FUNCTION_BLOCK EP7402_0xxx_Channel
VAR_INPUT
END_VAR
VAR_OUTPUT
END_VAR
VAR
	DI_Inputs AT%I* : DInputs;
	DO_Outputs AT%Q* : DOutputs;
	STM_Control AT%Q* : STMControl;
	STM_Info_data AT%I* : STMInfoData;
	STM_Input_Device AT%I* : STMInputDevice;
	STM_Status AT%I* : STMStatus;
	STM_Target_Velocity AT%Q* : STMTargetVelocity;
	
	_acceleration : UINT := 100;
	_deceleration : UINT := 100;
	
	State :(
		_00_mWait,
        _01_mReset,
        _02_mEnable,
		_03_mStop,
		_04_RunAtVelo,
		_05_mDisable);
		
	tonHoldHigh	: ton;
		
END_VAR

CASE State OF
        _00_mWait : 
			;
        _01_mReset : 
			STM_Control.reset := TRUE;
			tonHoldHigh(in := TRUE, pt := T#500MS);
			IF tonHoldHigh.Q THEN
				STM_Control.reset := FALSE;
				IF STM_Status.error = FALSE AND
					STM_Status.warning = FALSE AND
					STM_Status.ready = TRUE
				THEN
					State := _00_mWait;
					tonHoldHigh(in := FALSE);
				END_IF
			END_IF
			
        _02_mEnable : 
			IF STM_Status.error THEN				
				State := _01_mReset;
			ELSE
				STM_Control.enable := TRUE;			
			END_IF

			
		_04_RunAtVelo :
			;
			
		_03_mStop : 
			STM_Target_Velocity.velocity := 0;
			IF STM_Status.ready THEN	
				State := _02_mEnable;
			END_IF
			
		_05_mDisable:
			STM_Control.enable := FALSE;
			State := _00_mWait;
		
			
END_CASE

PROPERTY PUBLIC Acceleration : uint
GET
Acceleration := _acceleration;
END_GET
SET
_acceleration := Acceleration;
END_SET
END_PROPERTY

PROPERTY PUBLIC Deceleration : uint
GET
Deceleration := _deceleration;
END_GET
SET
_deceleration := Deceleration;
END_SET
END_PROPERTY

METHOD Disable : BOOL
VAR_INPUT
END_VAR
IF STM_Status.ready THEN
	State := _05_mDisable;
END_IF
END_METHOD

METHOD Enable : BOOL
VAR_INPUT
END_VAR
IF STM_Status.readyToEnable THEN
	State := _02_mEnable;
END_IF
END_METHOD

METHOD MoveNeg : BOOL
VAR_INPUT
END_VAR
STM_Control.invertDirection := TRUE;
STM_Target_Velocity.velocity := 6000;
STM_Target_Velocity.acceleration := _acceleration;
STM_Target_Velocity.deceleration := _deceleration;
State := _04_RunAtVelo;
END_METHOD

METHOD MovePos : BOOL
VAR_INPUT
END_VAR
STM_Control.invertDirection := FALSE;
STM_Target_Velocity.velocity := 6000;
STM_Target_Velocity.acceleration := _acceleration;
STM_Target_Velocity.deceleration := _deceleration;
State := _04_RunAtVelo;
END_METHOD

METHOD Reset : BOOL
VAR_INPUT
END_VAR
IF STM_Status.error OR STM_Status.warning THEN
	State := _01_mReset;
END_IF
END_METHOD

METHOD Stop : BOOL
VAR_INPUT
END_VAR
IF STM_Status.movingNegative OR STM_Status.movingPositive THEN
	State := _03_mStop;
END_IF
END_METHOD

END_FUNCTION_BLOCK

(* stored: Version 1.1.0.1, ProductVersion 3.1.4024.9
   POU EP7402_0xxx_Channel: Id {6c5f7c1d-1191-4da5-ba6c-9233e15b621c}, SpecialFunc None
   Property Acceleration: Id {fb806ad1-40c2-483b-8d67-b8b691be2e2e}
   Get Get: Id {695841d9-60cd-44a3-9a87-ad18a35882ea}
   Set Set: Id {0e599534-19e7-470a-b967-52a7758b8886}
   Property Deceleration: Id {7e1f896b-b060-403c-bef9-724c4b07da10}
   Get Get: Id {bd80b567-e82a-4c4f-9f77-142a6e2f190c}
   Set Set: Id {2b875229-85f0-47e3-80e3-932a5c73d028}
   Method Disable: Id {a3bf5df0-9c23-4707-adfd-85b9fcedd433}
   Method Enable: Id {69b44551-5844-42d2-b1fb-69cd7479da38}
   Method MoveNeg: Id {b2140de2-50ba-45d3-8d0c-e25d3c8c6c62}
   Method MovePos: Id {cfec3af2-c578-4937-a526-cc8a734135af}
   Method Reset: Id {27080227-2c5a-4495-a769-d9715d06fcf4}
   Method Stop: Id {cf5a21b5-0585-43bb-ad8d-f1808560a28e} *)
